FUNCTION_BLOCK ThreeConCtl (* Composite Function Block Type *)
  (* Standard: 61499-2 *)
  (* Version 0.2, 2003-12-05, JHC, Rockwell Automation, Renamed from NEWCOMPFB. *)
  (* Version 0.1, 2002-01-08, JHC, Rockwell Automation, Added DLY FB as example. *)
  (* Version 0.0, 2000-05-27, JHC, Rockwell Automation *)
  (* Compiler header: package fb.rt.cs725; *)
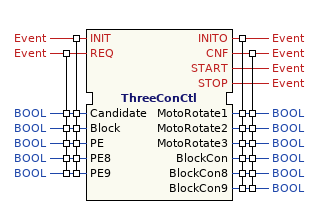
  EVENT_INPUT
    INIT WITH Candidate, Block, PE, PE8, PE9; (* Initialization Request *)
    REQ WITH Block, Candidate, PE, PE9, PE8; (* Normal Execution Request *)
  END_EVENT
  EVENT_OUTPUT
    INITO WITH MotoRotate1, MotoRotate2, MotoRotate3, BlockCon, BlockCon9, BlockCon8; (* Initialization Confirm *)
    CNF WITH MotoRotate1, MotoRotate2, MotoRotate3, BlockCon, BlockCon8, BlockCon9; (* Execution Confirmation *)
    START;
    STOP;
  END_EVENT
  VAR_INPUT
    Candidate : BOOL;
    Block : BOOL;
    PE : BOOL;
    PE8 : BOOL;
    PE9 : BOOL;
  END_VAR
  VAR_OUTPUT
    MotoRotate1 : BOOL;
    MotoRotate2 : BOOL;
    MotoRotate3 : BOOL;
    BlockCon : BOOL;
    BlockCon8 : BOOL;
    BlockCon9 : BOOL;
  END_VAR
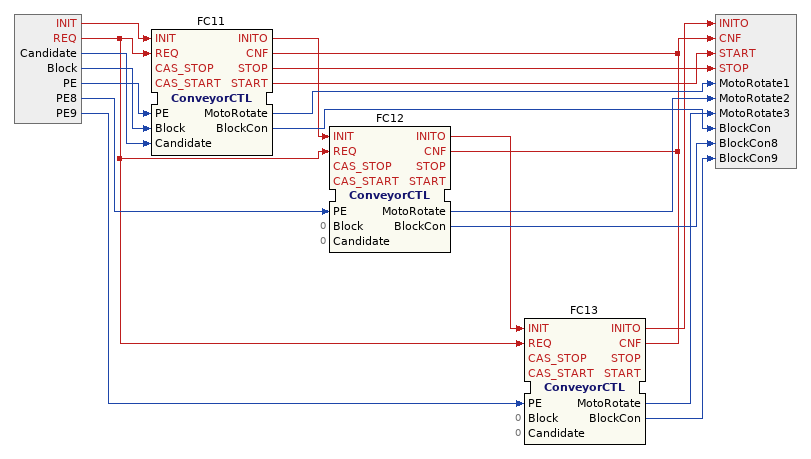
  FBS
    FC11 : ConveyorCTL;
    FC12 : ConveyorCTL(Block := 0, Candidate := 0);
    FC13 : ConveyorCTL(Block := 0, Candidate := 0);
  END_FBS
  EVENT_CONNECTIONS
    INIT TO FC11.INIT;
    REQ TO FC11.REQ;
    FC11.INITO TO FC12.INIT;
    FC12.INITO TO FC13.INIT;
    FC13.INITO TO INITO;
    FC13.CNF TO CNF;
    FC11.STOP TO STOP;
    FC11.START TO START;
    REQ TO FC12.REQ;
    REQ TO FC13.REQ;
    FC11.CNF TO CNF;
    FC12.CNF TO CNF;
  END_CONNECTIONS
  DATA_CONNECTIONS
    FC13.MotoRotate TO MotoRotate3;
    FC12.MotoRotate TO MotoRotate2;
    FC11.MotoRotate TO MotoRotate1;
    PE TO FC11.PE;
    Block TO FC11.Block;
    FC11.BlockCon TO BlockCon;
    Candidate TO FC11.Candidate;
    PE8 TO FC12.PE;
    PE9 TO FC13.PE;
    FC13.BlockCon TO BlockCon9;
    FC12.BlockCon TO BlockCon8;
  END_CONNECTIONS
END_FUNCTION_BLOCK
